(* PLC project Unnamed, Unknown Unnamed 1 *)
(* stored: creationDateTime 2022-08-16T15:49:17, modificationDateTime 2024-10-15T13:02:18 *)

PROGRAM PLC_STEP_PULSE_CTR
  VAR_EXTERNAL
    position_motor1_1 : DWORD;
    position_motor2_1 : DWORD;
    position_motor3_1 : DWORD;
    position_motor4_1 : DWORD;
    position_motor5_1 : DWORD;
    position_motor6_1 : DWORD;
    position_motor7_1 : DWORD;
    position_motor8_1 : DWORD;
  END_VAR
  VAR
    step_1 : DWORD;
    step_2 : DWORD;
    step_3 : DWORD;
    step_4 : DWORD;
    step_5 : DWORD;
    step_6 : DWORD;
    step_7 : DWORD;
    step_8 : DWORD;
    en_motor1 : BOOL;
    en_motor2 : BOOL;
    en_motor3 : BOOL;
    en_motor4 : BOOL;
    en_motor5 : BOOL;
    en_motor6 : BOOL;
    en_motor7 : BOOL;
    en_motor8 : BOOL;
  END_VAR
  VAR_EXTERNAL
    cw_m1 : BOOL;
    cw_m2 : BOOL;
    cw_m3 : BOOL;
    cw_m4 : BOOL;
    cw_m5 : BOOL;
    cw_m6 : BOOL;
    cw_m7 : BOOL;
    cw_m8 : BOOL;
    ccw_m1 : BOOL;
    ccw_m2 : BOOL;
    ccw_m3 : BOOL;
    ccw_m4 : BOOL;
    ccw_m5 : BOOL;
    ccw_m6 : BOOL;
    ccw_m7 : BOOL;
    ccw_m8 : BOOL;
  END_VAR
  VAR
    ccw_m1_on : BOOL;
    ccw_m2_on : BOOL;
    ccw_m3_on : BOOL;
    ccw_m4_on : BOOL;
    ccw_m5_on : BOOL;
    ccw_m6_on : BOOL;
    ccw_m7_on : BOOL;
    ccw_m8_on : BOOL;
    cw_m1_on : BOOL;
    cw_m2_on : BOOL;
    cw_m3_on : BOOL;
    cw_m4_on : BOOL;
    cw_m5_on : BOOL;
    cw_m6_on : BOOL;
    cw_m7_on : BOOL;
    cw_m8_on : BOOL;
  END_VAR
  VAR_EXTERNAL
    data_moto1 : BYTE;
    data_moto2 : BYTE;
    data_moto3 : BYTE;
    data_moto4 : BYTE;
    data_moto5 : BYTE;
    data_moto6 : BYTE;
    data_moto7 : BYTE;
    data_moto8 : BYTE;
    current_M1_pos : DWORD;
    current_M2_pos : DWORD;
    current_M3_pos : DWORD;
    current_M4_pos : DWORD;
    current_M5_pos : DWORD;
    current_M6_pos : DWORD;
    current_M7_pos : DWORD;
    current_M8_pos : DWORD;
  END_VAR
  VAR
    current_1_vitri : DWORD;
    current_2_vitri : DWORD;
    current_3_vitri : DWORD;
    current_4_vitri : DWORD;
    current_5_vitri : DWORD;
    current_6_vitri : DWORD;
    current_7_vitri : DWORD;
    current_8_vitri : DWORD;
  END_VAR
  VAR_EXTERNAL
    motor1_speed : UINT;
    motor2_speed : UINT;
    motor3_speed : UINT;
    motor4_speed : UINT;
    motor5_speed : UINT;
    motor6_speed : UINT;
    motor7_speed : UINT;
    motor8_speed : UINT;
  END_VAR
  VAR
    set_motor1_speed : UINT := 8000;
    set_motor2_speed : UINT := 8000;
    set_motor3_speed : UINT := 8000;
    set_motor4_speed : UINT := 8000;
    set_motor5_speed : UINT := 8000;
    set_motor6_speed : UINT := 8000;
    set_motor7_speed : UINT := 8000;
    set_motor8_speed : UINT := 8000;
    set_motor1_accel : UINT := 2000;
    set_motor2_accel : UINT := 2000;
    set_motor3_accel : UINT := 2000;
    set_motor4_accel : UINT := 2000;
    set_motor5_accel : UINT := 2000;
    set_motor6_accel : UINT := 2000;
    set_motor7_accel : UINT := 2000;
    set_motor8_accel : UINT := 2000;
  END_VAR
  VAR_EXTERNAL
    motor1_accel : UINT;
    motor2_accel : UINT;
    motor3_accel : UINT;
    motor4_accel : UINT;
    motor5_accel : UINT;
    motor6_accel : UINT;
    motor7_accel : UINT;
    motor8_accel : UINT;
  END_VAR
  VAR
    mode_run_m1 : BYTE;
    mode_run_m2 : BYTE;
    mode_run_m3 : BYTE;
    mode_run_m4 : BYTE;
    mode_run_m5 : BYTE;
    mode_run_m6 : BYTE;
    mode_run_m7 : BYTE;
    mode_run_m8 : BYTE;
  END_VAR
  VAR_EXTERNAL
    START_Moto_1 : BOOL;
    START_Moto_2 : BOOL;
    START_Moto_3 : BOOL;
    START_Moto_4 : BOOL;
    START_Moto_5 : BOOL;
    START_Moto_6 : BOOL;
    START_Moto_7 : BOOL;
    START_Moto_8 : BOOL;
    motor1_running : BOOL;
    motor2_running : BOOL;
    motor3_running : BOOL;
    motor4_running : BOOL;
    motor5_running : BOOL;
    motor6_running : BOOL;
    motor7_running : BOOL;
    motor8_running : BOOL;
    motor1_position_ok : BOOL;
    motor2_position_ok : BOOL;
    motor3_position_ok : BOOL;
    motor4_position_ok : BOOL;
    motor5_position_ok : BOOL;
    motor6_position_ok : BOOL;
    motor7_position_ok : BOOL;
    motor8_position_ok : BOOL;
  END_VAR
  VAR
    MOTOR1_RUNING : BOOL;
    MOTOR2_RUNING : BOOL;
    MOTOR3_RUNING : BOOL;
    MOTOR4_RUNING : BOOL;
    MOTOR5_RUNING : BOOL;
    MOTOR6_RUNING : BOOL;
    MOTOR7_RUNING : BOOL;
    MOTOR8_RUNING : BOOL;
    MOTOR1_POS_ok : BOOL;
    MOTOR2_POS_ok : BOOL;
    MOTOR3_POS_ok : BOOL;
    MOTOR4_POS_ok : BOOL;
    MOTOR5_POS_ok : BOOL;
    MOTOR6_POS_ok : BOOL;
    MOTOR7_POS_ok : BOOL;
    MOTOR8_POS_ok : BOOL;
  END_VAR
  VAR_EXTERNAL
    zero_m1_kaki_ok : BOOL;
    zero_m2_kaki_ok : BOOL;
    zero_m3_kaki_ok : BOOL;
    zero_m4_kaki_ok : BOOL;
    zero_m5_kaki_ok : BOOL;
    zero_m6_kaki_ok : BOOL;
    zero_m7_kaki_ok : BOOL;
    zero_m8_kaki_ok : BOOL;
  END_VAR

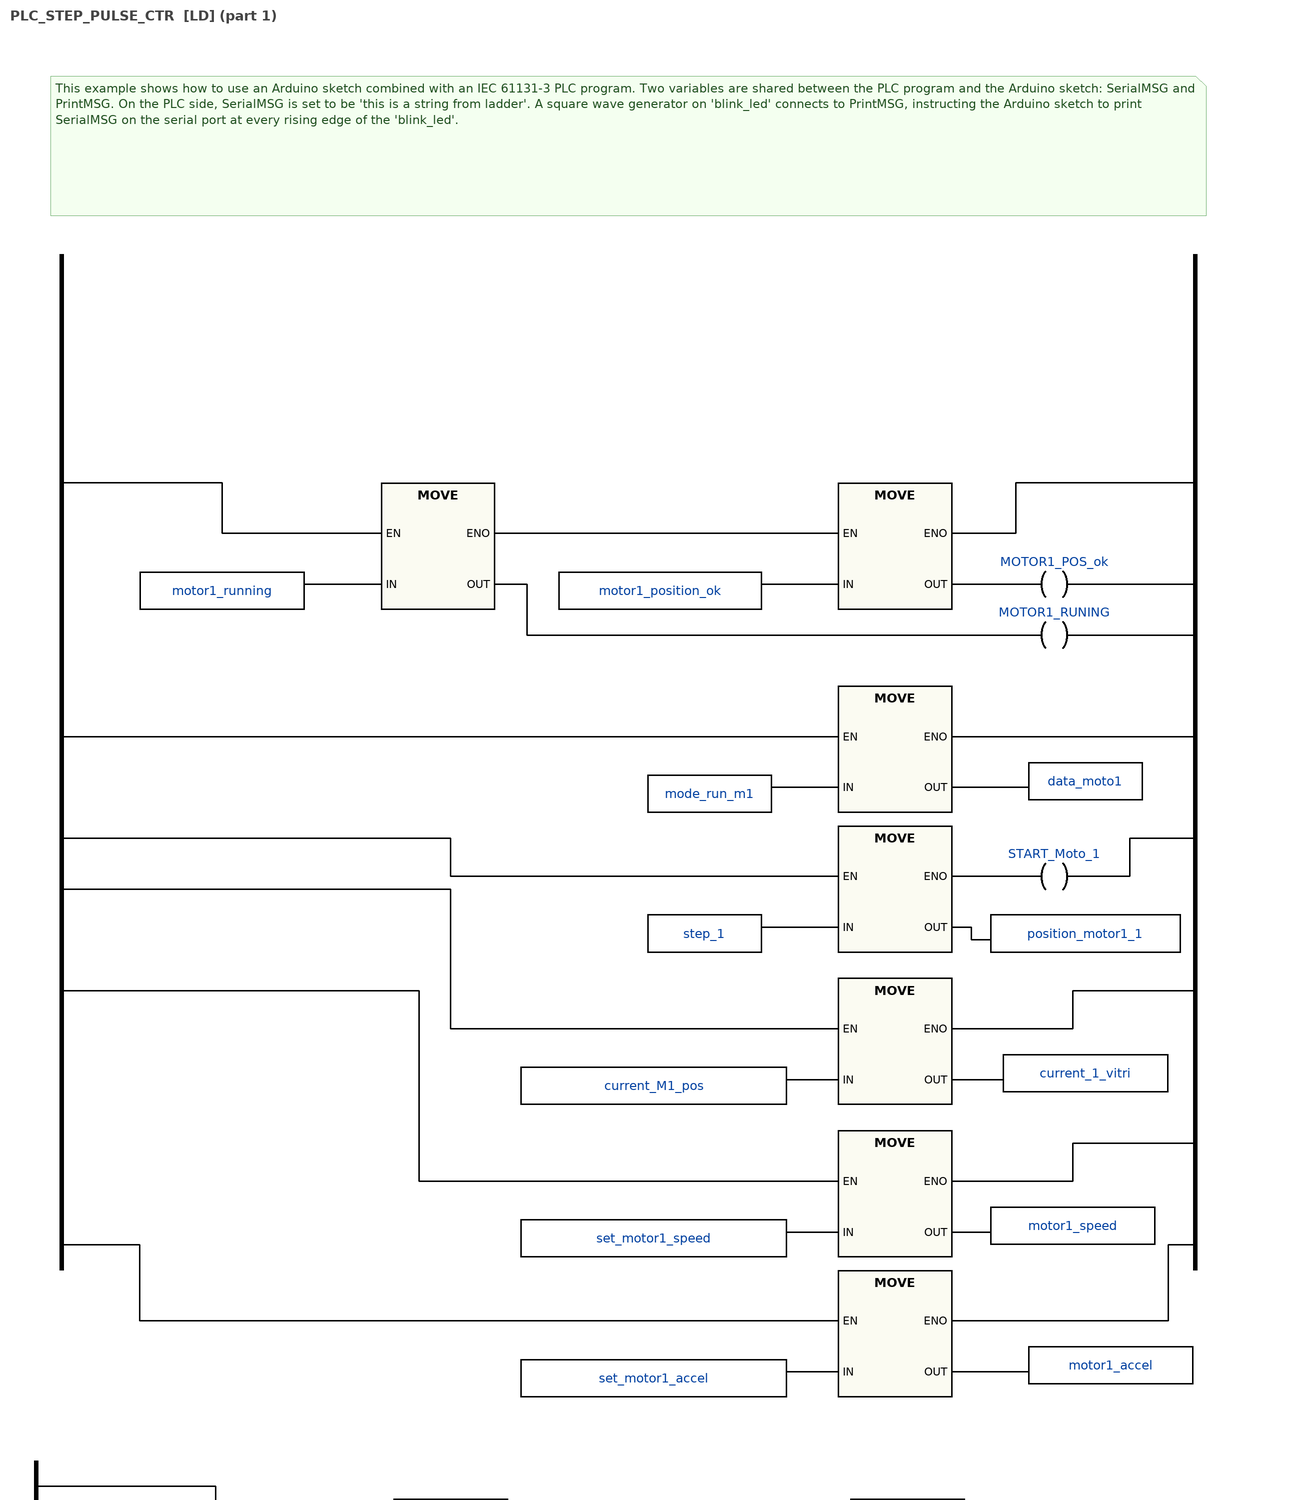
(* LD diagram, written out as Structured Text *)
(* This example shows how to use an Arduino sketch combined with an IEC 61131-3 PLC program. Two variables are shared between the PLC program and the Arduino sketch: SerialMSG and PrintMSG. On the PLC side, SerialMSG is set to be 'this is a string from ladder'. A square wave generator on 'blink_led' connects to PrintMSG, instructing the Arduino sketch to print SerialMSG on the serial port at every rising edge of the 'blink_led'. *)
position_motor1_1 := step_1;
data_moto1 := mode_run_m1;
current_1_vitri := current_M1_pos;
motor1_speed := set_motor1_speed;
motor1_accel := set_motor1_accel;
START_Moto_1 := TRUE;
MOTOR1_POS_ok := motor1_position_ok;
MOTOR1_RUNING := motor1_running;
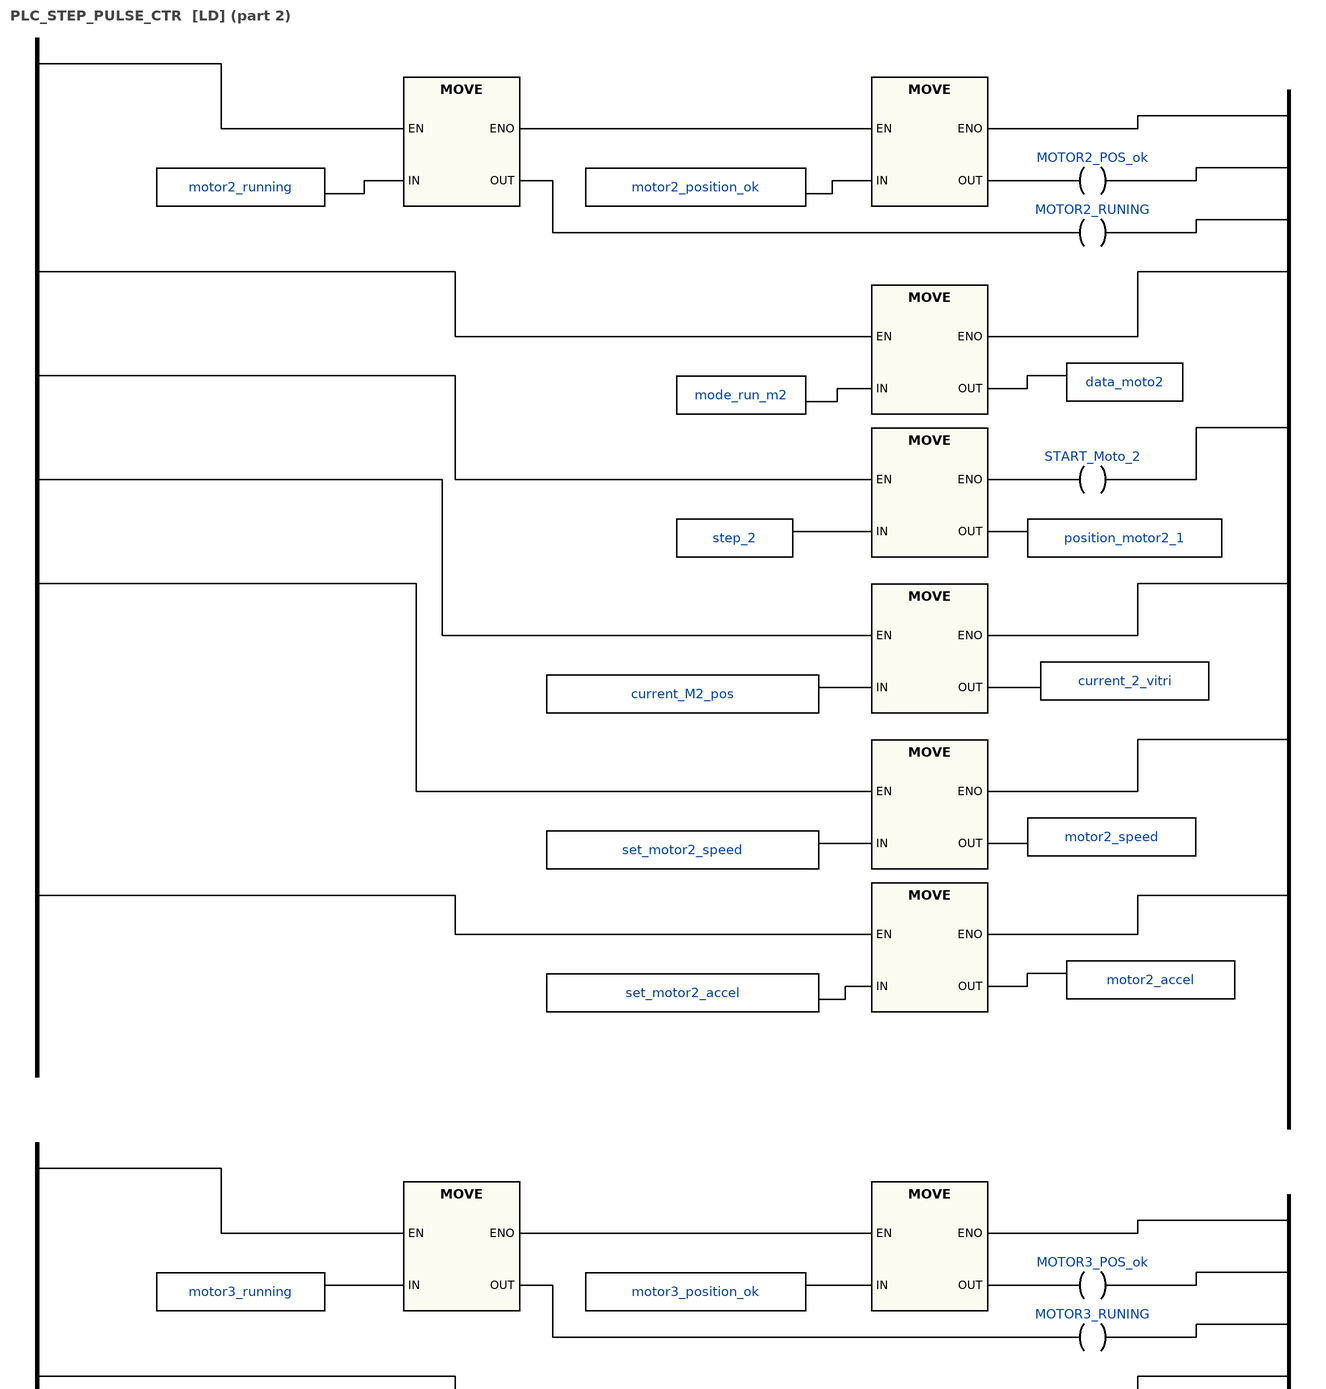
MOTOR2_POS_ok := motor2_position_ok;
MOTOR2_RUNING := motor2_running;
START_Moto_2 := TRUE;
position_motor2_1 := step_2;
data_moto2 := mode_run_m2;
current_2_vitri := current_M2_pos;
motor2_speed := set_motor2_speed;
motor2_accel := set_motor2_accel;
MOTOR3_POS_ok := motor3_position_ok;
MOTOR3_RUNING := motor3_running;
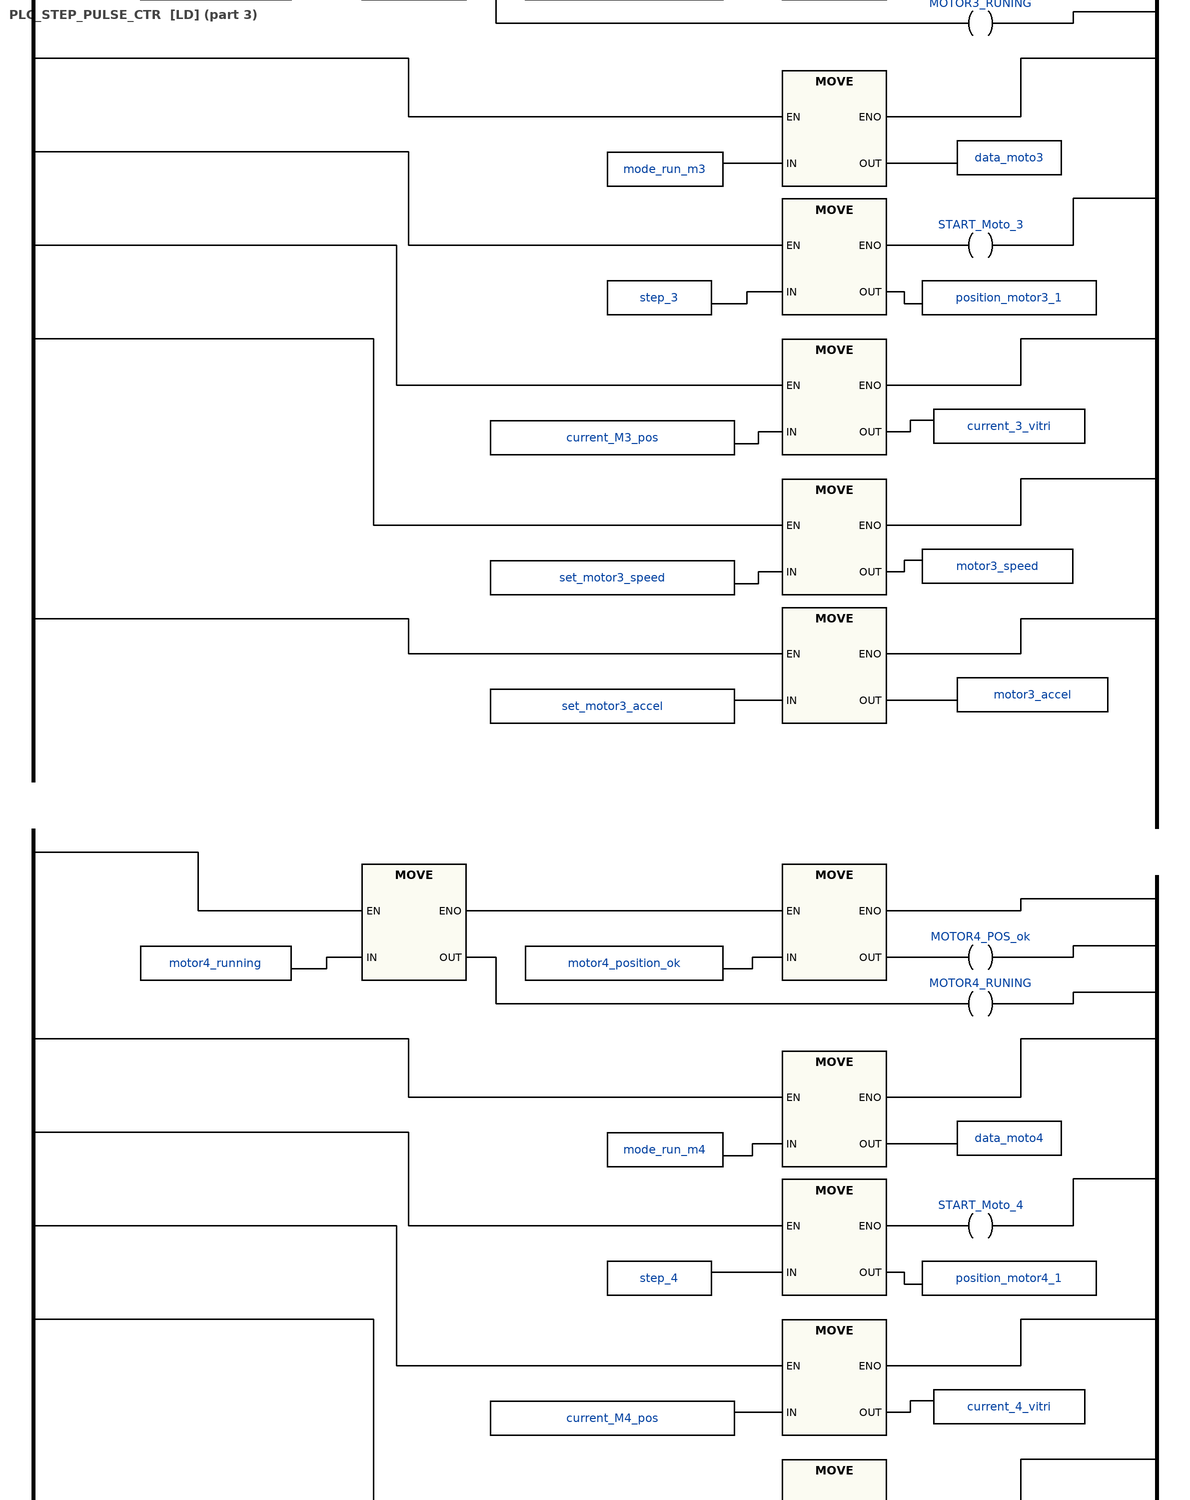
START_Moto_3 := TRUE;
position_motor3_1 := step_3;
data_moto3 := mode_run_m3;
current_3_vitri := current_M3_pos;
motor3_speed := set_motor3_speed;
motor3_accel := set_motor3_accel;
MOTOR4_POS_ok := motor4_position_ok;
MOTOR4_RUNING := motor4_running;
START_Moto_4 := TRUE;
position_motor4_1 := step_4;
data_moto4 := mode_run_m4;
current_4_vitri := current_M4_pos;
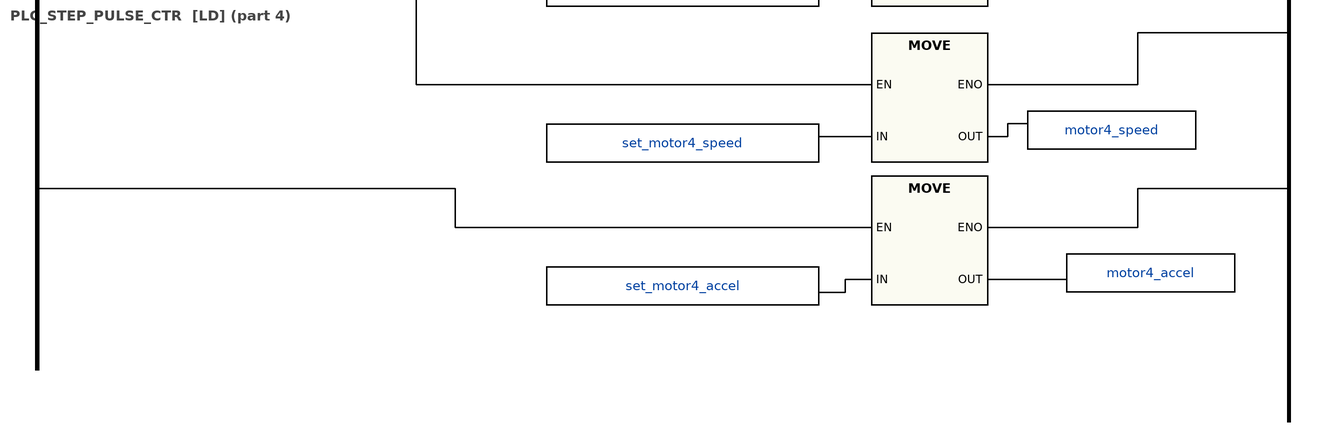
motor4_speed := set_motor4_speed;
motor4_accel := set_motor4_accel;
END_PROGRAM

PROGRAM main
  VAR
    TOF0 : TOF;
    TON0 : TON;
  END_VAR
  VAR
    blink_led0 AT %QX0.0 : BOOL;
    blink_led1 AT %QX0.1 : BOOL;
    blink_led2 AT %QX6.3 : BOOL;
  END_VAR
  VAR
    blink_led3 : BOOL;
  END_VAR
  VAR
    blink_led4 AT %QX0.4 : BOOL;
    blink_led5 AT %QX0.5 : BOOL;
    blink_led6 AT %QX0.6 : BOOL;
    blink_led7 AT %QX0.7 : BOOL;
    Analog_A0 AT %IW0 : INT;
    Analog_A1 AT %IW1 : INT;
    Analog_A2 AT %IW2 : INT;
    Analog_A3 AT %IW3 : INT;
  END_VAR
  VAR
    Analog_A0_value : INT;
    Analog_A1_value : INT;
    Analog_A2_value : INT;
    Analog_A3_value : INT;
  END_VAR
  VAR
    button0 AT %IX0.0 : BOOL;
    button1 AT %IX0.1 : BOOL;
    button2 AT %IX0.2 : BOOL;
    button3 AT %IX0.3 : BOOL;
  END_VAR
  VAR
    button_tem0 : BOOL;
    button_tem1 : BOOL;
    button_tem2 : BOOL;
    button_tem3 : BOOL;
  END_VAR
  VAR
    blink_led8 AT %QX1.0 : BOOL;
    blink_led9 AT %QX1.1 : BOOL;
    blink_led10 AT %QX1.2 : BOOL;
    blink_led11 AT %QX1.3 : BOOL;
  END_VAR
  VAR_OUTPUT
    temp_coil : BOOL;
    temp_coil0 : BOOL;
  END_VAR
  VAR_INPUT
    temp_BT : BOOL;
    temp_BT0 : BOOL;
  END_VAR
  VAR_EXTERNAL
    lr_0 : BOOL;
    lr_1 : BOOL;
    lr_2 : BOOL;
    lr_3 : BOOL;
    lr_4 : BOOL;
    lr_5 : BOOL;
    lr_6 : BOOL;
    lr_7 : BOOL;
    lr_8 : BOOL;
    lr_9 : BOOL;
    lr_10 : BOOL;
    lr_11 : BOOL;
    lr_12 : BOOL;
    lr_13 : BOOL;
    lr_14 : BOOL;
    lr_15 : BOOL;
    dm_0 : DWORD;
    dm_1 : DWORD;
    dm_2 : DWORD;
    dm_3 : DWORD;
    dm_4 : DWORD;
    dm_5 : DWORD;
    dm_6 : DWORD;
    dm_7 : DWORD;
    dm_8 : DWORD;
    dm_9 : DWORD;
    dm_10 : DWORD;
    dm_11 : DWORD;
    dm_12 : DWORD;
    dm_13 : DWORD;
    dm_14 : DWORD;
    dm_15 : DWORD;
    dm_16 : DWORD;
    dm_17 : DWORD;
    dm_18 : DWORD;
    dm_19 : DWORD;
  END_VAR
  VAR
    temp_1 : DWORD;
    temp_2 : DWORD;
    temp_3 : DWORD;
    temp_4 : DWORD;
    temp_5 : DWORD;
    temp_6 : DWORD;
    temp_7 : DWORD;
    test : BOOL;
    test0 : DWORD;
    test1 : DWORD;
    test2 : DWORD;
    test3 : DWORD;
    test4 : DWORD;
    test5 : DWORD;
    test6 : DWORD;
    test7 : DWORD;
    coil_lr : BOOL;
    coil_lr0 : BOOL;
    coil_lr1 : BOOL;
    coil_lr2 : BOOL;
    coil_lr3 : BOOL;
  END_VAR
  VAR_EXTERNAL
    coil_256 : UINT;
  END_VAR
  VAR
    coil_257 : UINT;
  END_VAR

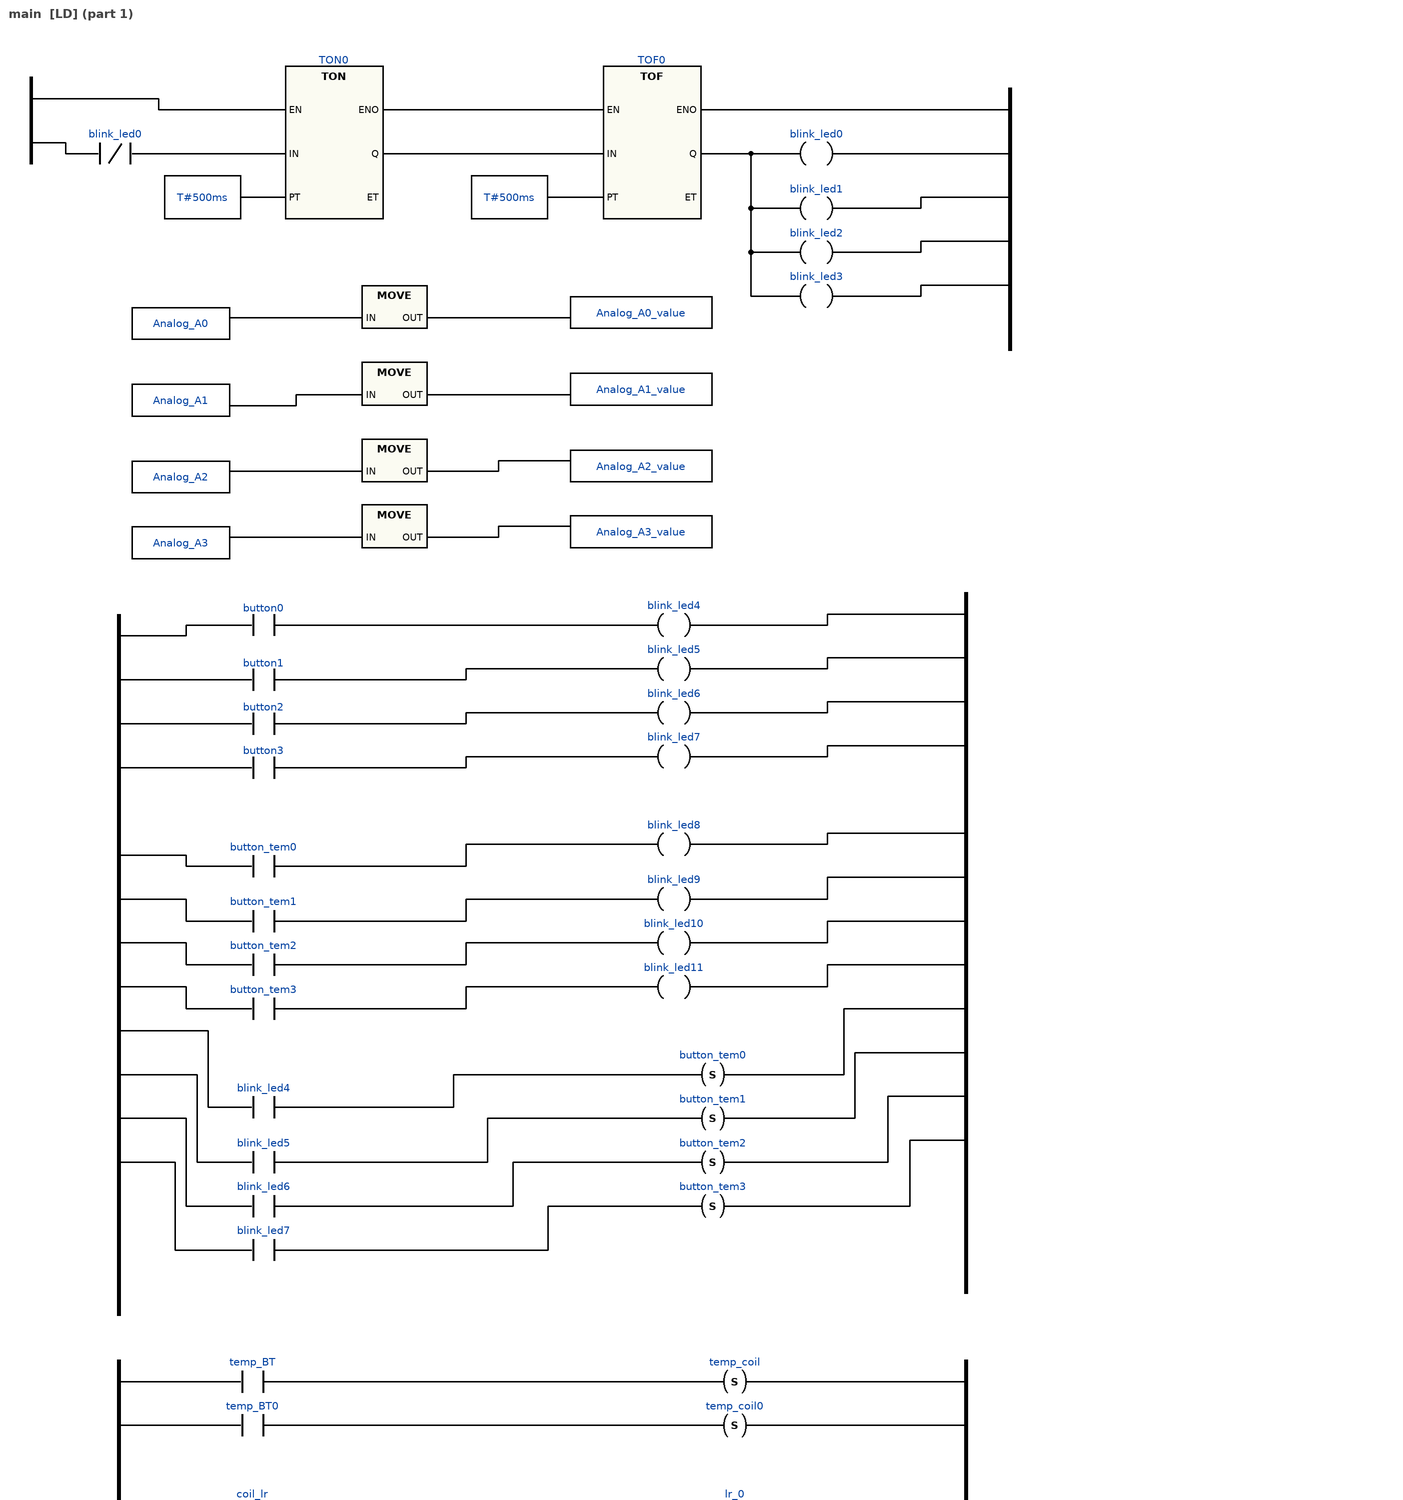
(* LD diagram, written out as Structured Text *)
TON0(IN := NOT blink_led0, PT := T#500ms);
TOF0(EN := TON0.ENO, IN := TON0.Q, PT := T#500ms);
blink_led0 := TOF0.Q;
Analog_A0_value := Analog_A0;
Analog_A1_value := Analog_A1;
Analog_A2_value := Analog_A2;
Analog_A3_value := Analog_A3;
blink_led1 := TOF0.Q;
blink_led2 := TOF0.Q;
blink_led3 := TOF0.Q;
blink_led4 := button0;
blink_led5 := button1;
blink_led6 := button2;
blink_led7 := button3;
blink_led8 := button_tem0;
blink_led9 := button_tem1;
blink_led10 := button_tem2;
blink_led11 := button_tem3;
IF blink_led4 THEN button_tem0 := TRUE; END_IF;
IF blink_led5 THEN button_tem1 := TRUE; END_IF;
IF blink_led6 THEN button_tem2 := TRUE; END_IF;
IF blink_led7 THEN button_tem3 := TRUE; END_IF;
IF temp_BT THEN temp_coil := TRUE; END_IF;
IF temp_BT0 THEN temp_coil0 := TRUE; END_IF;
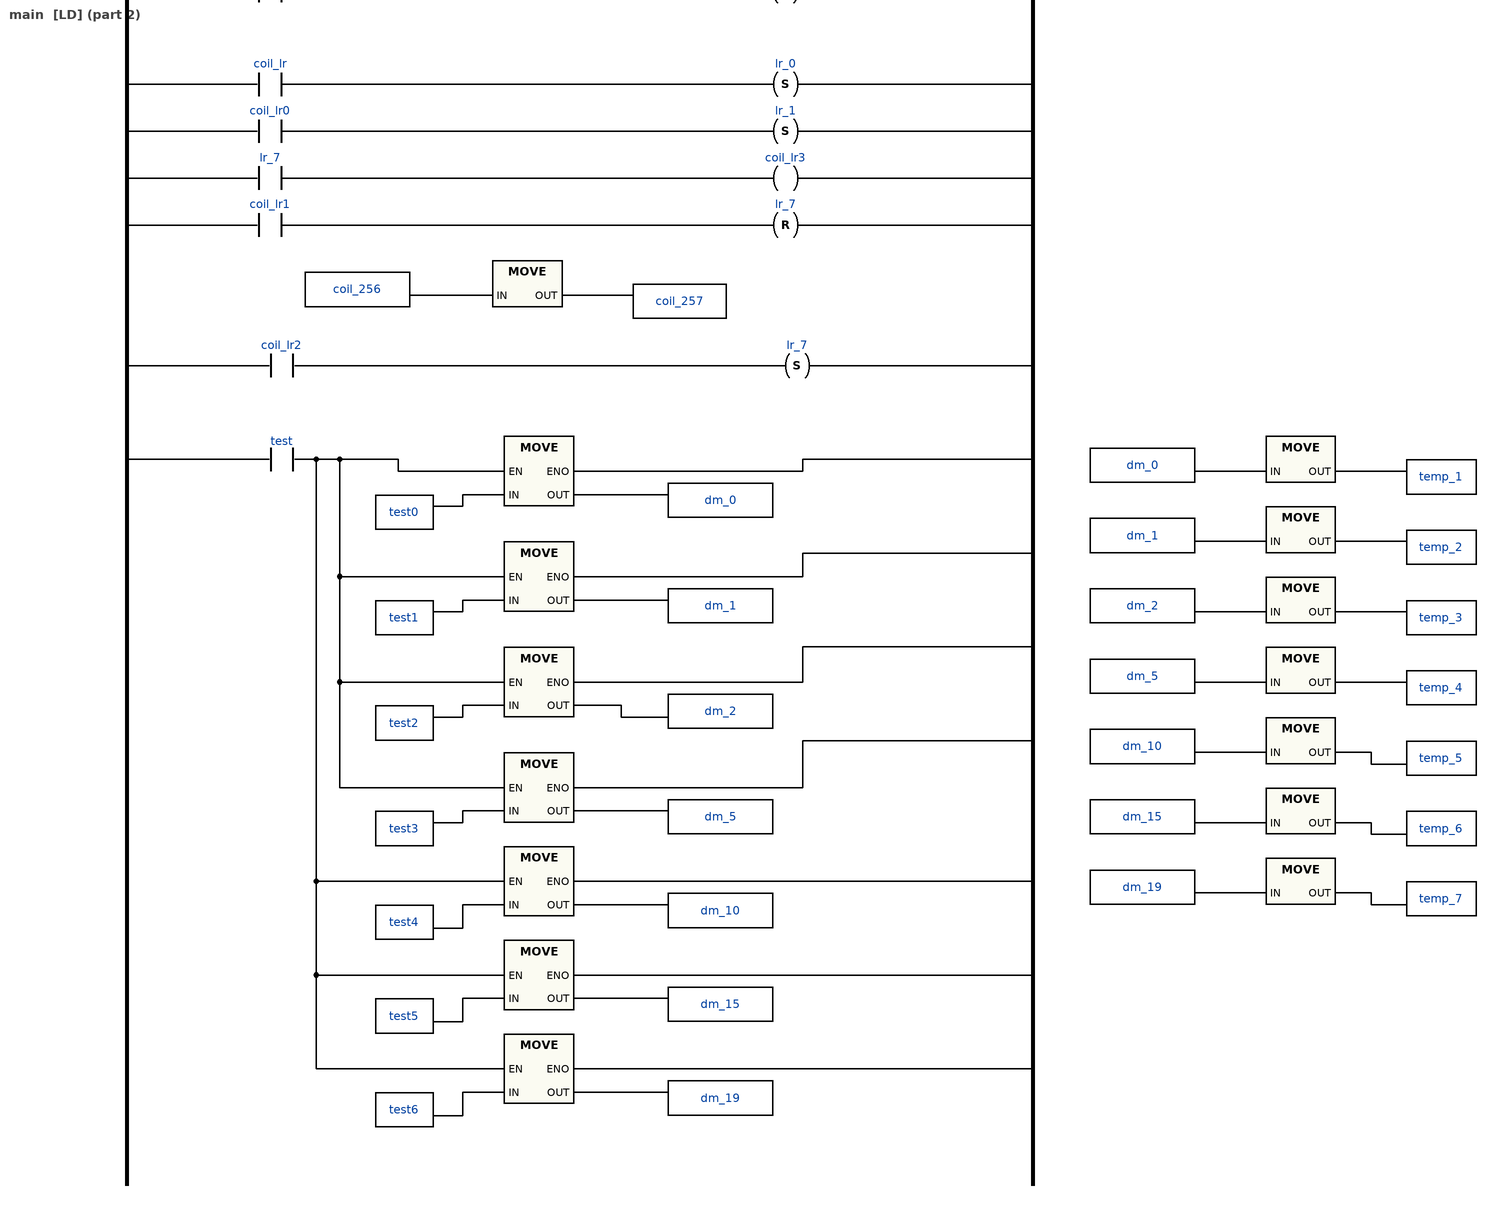
temp_1 := dm_0;
temp_2 := dm_1;
temp_3 := dm_2;
temp_4 := dm_5;
IF test THEN dm_0 := test0; END_IF;
IF test THEN dm_1 := test1; END_IF;
IF test THEN dm_2 := test2; END_IF;
IF test THEN dm_5 := test3; END_IF;
IF test THEN dm_10 := test4; END_IF;
IF test THEN dm_15 := test5; END_IF;
IF test THEN dm_19 := test6; END_IF;
temp_5 := dm_10;
temp_6 := dm_15;
temp_7 := dm_19;
IF coil_lr THEN lr_0 := TRUE; END_IF;
IF coil_lr0 THEN lr_1 := TRUE; END_IF;
coil_lr3 := lr_7;
coil_257 := coil_256;
IF coil_lr1 THEN lr_7 := FALSE; END_IF;
IF coil_lr2 THEN lr_7 := TRUE; END_IF;
END_PROGRAM

CONFIGURATION Config0
  RESOURCE Res0 ON PLC
    TASK task0(INTERVAL := T#5ms, PRIORITY := 0);
    TASK task1(INTERVAL := T#10ms, PRIORITY := 0);
    PROGRAM instance0 WITH task0 : PLC_STEP_PULSE_CTR;
    PROGRAM instance1 WITH task1 : main;
  END_RESOURCE
END_CONFIGURATION
